FUNCTION WRITE_PROTECTED_WSTRING
VAR_INPUT
    Ptr : POINTER TO WSTRING;
    Value : WSTRING;
END_VAR

Ptr^ := Value;

END_FUNCTION

(* stored: Version 1.1.0.1
   POU WRITE_PROTECTED_WSTRING: Id {d2b8e71b-44e5-4ea8-8ec3-be2deccd6175}, SpecialFunc None *)
